// TIA Portal V17 export
// export: Created 2025-08-05T09:36:00.4673777Z, ExportSetting WithDefaults, DisplayName Totally Integrated Automation Portal, DisplayVersion V17, DisplayName TIA Portal Openness, DisplayVersion V17, DisplayName TIA Portal Version Control Interface, DisplayVersion V17, DisplayName SINAMICS Startdrive Advanced, DisplayVersion V17, DisplayName SINAMICS Startdrive G130, G150, S120, S150, SINAMICS MV, S210, DisplayVersion V17, DisplayName SINAMICS Startdrive G110M, G120, G120C, G120D, G120P, G115D, DisplayVersion V17, DisplayName STEP 7 Professional, DisplayVersion V17, DisplayName STEP 7 Safety, DisplayVersion V17, DisplayName WinCC Advanced, DisplayVersion V17
TYPE "typeHmiUserManagement"
TITLE = HMI user management / HMI Benutzerverwaltung
// HMI user management [V 01.00 | Kernel_V2] / HMI Benutzerverwaltung [V 01.00 | Kernel_V2]
// stored: IsFailsafeCompliant false
   STRUCT
      activeUserLevel : "typeUserLevel";   // Benutzerlevel / User level
      eks : Struct   // EKS Protection Level / EKS protection level
         protectionLevel : Int;   // Ausgabe der Schutzstufe / Output of protection level
         checksumNok : Bool;   // EKS Checksumme des Schlüssels n.i.O. / EKS check sum of key NOK
         dateNok : Bool;   // EKS Ablaufdatum des Schlüssels n.i.O. / EKS expiry data of key NOK
         costCenterNok : Bool;   // EKS Kostenstelle des Schlüssels n.i.O. / EKs cost center of key NOK
         eksKeyInvalidLess30Days : Bool;   // EKS Schlüssel wird in 30 Tagen ungültig / EKS key will expire in 30 days
         eksAdapterReady : Bool;   // EKS Adapter betriebsbereit / EKS adapter ready for operation
         eksKeyDetected : Bool;   // EKS Schlüssel erkannt / EKS key detected
         operatiorId : Int;   // EKS Operator ID / EKS operator ID
      END_STRUCT;
   END_STRUCT;
END_TYPE
